FUNCTION_BLOCK INTERNAL FB_Autumn EXTENDS FB_SeasonBase
VAR_INPUT
END_VAR
VAR_OUTPUT
END_VAR
VAR
END_VAR

METHOD FB_init : BOOL
VAR_INPUT
    bInitRetains:           BOOL; // if TRUE, the retain variables are initialized (warm start / cold start)
    bInCopyCode:            BOOL;  // if TRUE, the instance afterwards gets moved into the copy code (online change)
    ipStateMachine:         I_StateMachine;
    ipParentObject:         I_Object;
END_VAR
THIS^._eState := E_Season.Autumn;
END_METHOD

METHOD  NextSeason
VAR_INPUT
END_VAR
THIS^.ipStateMachine.SetState(THIS^.ipSeasonCtrl.StateWinter);
END_METHOD

METHOD OnEntry
VAR_INPUT
END_VAR
SUPER^.OnEntry();
THIS^._bWindBlowing     := TRUE;
THIS^._bRaining         := FALSE;
THIS^._bSunShining      := FALSE;
THIS^._bSnowing         := FALSE;
THIS^._nLeavesState     := 2;

Tc2_System.ADSLOGSTR(msgCtrlMask := THIS^._nLogLevel,
                     msgFmtStr := 'Leaves are changing color to yellow/orange/bright red',
                     strArg := '');
END_METHOD

METHOD OnExit
SUPER^.OnExit();
THIS^._bWindBlowing     := FALSE;
THIS^._bRaining         := FALSE;
THIS^._bSunShining      := FALSE;
THIS^._bSnowing         := FALSE;
THIS^._nLeavesState     := 2;
END_METHOD

END_FUNCTION_BLOCK

(* stored: Version 1.1.0.1, ProductVersion 3.1.4024.12
   POU FB_Autumn: Id {3c70ed3c-2964-07ba-0255-0adc2cfa14bd}, SpecialFunc None
   Method FB_init: Id {1fcc3135-6dfb-0f70-317b-3513f07762dd}
   Method NextSeason: Id {3484f1e5-681a-0edc-0024-bb82b9308abf}
   Method OnEntry: Id {5d8a78bf-6c5e-0b9d-3494-52e82bbf9a3d}
   Method OnExit: Id {04a54a9c-a721-0dc6-39ec-e6fb88250a75} *)
